(*$
<p>This function configures a generic <a target="_blank" href="#iol_slave">iol_slave</a> as a <strong>Sick WTB2SC - 2P3244</strong>. It allow to connect the object to the device-specific
parameters structure variable <a target="_blank" href="#iol_slave_wtb2sc_data">iol_slave_wtb2sc_data</a>.</p>
<p>This function should be called at startup only.</p>
$*)

FUNCTION iol_slave_mlg2prime_configure : VOID
VAR_IN_OUT
	data:						iol_slave_mlg2prime_data;			(*$	Parameters struct variable$*)
	CONVERSION_this:						iol_slave;						(*$ Instance to which the method applies $*)
END_VAR

VAR CONSTANT
	NULL:                                   			XWORD := 0;
END_VAR

//IF iol_slave_is_not_initialized(CONVERSION_this := CONVERSION_this)
//	OR
IF	iol_slave_is_configured(CONVERSION_this := CONVERSION_this)
THEN
	RETURN;
END_IF

(*** Start parameter configuration ***)

(* STANDARD PARAMETERS CONFIGURATION *)

iol_slave_configure_parameter(
	current_value_address := ADR(CONVERSION_this.vendor_name),
	configured_value_address := NULL,
	length := SIZEOF(CONVERSION_this.vendor_name),
	_type := ADST_STRING,
	coe_index := 16#0010,
	coe_sub_index := 16#00,
	readable := TRUE,
	writeable := FALSE,
	to_check := FALSE,
	CONVERSION_this := CONVERSION_this);

iol_slave_configure_parameter(
	current_value_address := ADR(CONVERSION_this.product_name),
	configured_value_address := NULL,
	length := SIZEOF(CONVERSION_this.product_name),
	_type := ADST_STRING,
	coe_index := 16#0012,
	coe_sub_index := 16#00,
	readable := TRUE,
	writeable := FALSE,
	to_check := FALSE,
	CONVERSION_this := CONVERSION_this);

iol_slave_configure_parameter(
	current_value_address := ADR(CONVERSION_this.product_id),
	configured_value_address := NULL,
	length := SIZEOF(CONVERSION_this.product_id),
	_type := ADST_STRING,
	coe_index := 16#0013,
	coe_sub_index := 16#00,
	readable := TRUE,
	writeable := FALSE,
	to_check := FALSE,
	CONVERSION_this := CONVERSION_this);


iol_slave_configure_parameter(
	current_value_address := ADR(CONVERSION_this.hardware_revision),
	configured_value_address := NULL,
	length := SIZEOF(CONVERSION_this.hardware_revision),
	_type := ADST_STRING,
	coe_index := 16#0016,
	coe_sub_index := 16#00,
	readable := TRUE,
	writeable := FALSE,
	to_check := FALSE,
	CONVERSION_this := CONVERSION_this);

iol_slave_configure_parameter(
	current_value_address := ADR(CONVERSION_this.firmware_revision),
	configured_value_address := NULL,
	length := SIZEOF(CONVERSION_this.firmware_revision),
	_type := ADST_STRING,
	coe_index := 16#0017,
	coe_sub_index := 16#00,
	readable := TRUE,
	writeable := FALSE,
	to_check := FALSE,
	CONVERSION_this := CONVERSION_this);


(* CUSTOM PARAMETERS CONFIGURATION *)


iol_slave_configure_parameter(
	current_value_address := ADR(data.CrossBeamEnable),
	configured_value_address := ADR(data.CrossBeamEnable),
	length := SIZEOF(data.CrossBeamEnable),
	_type := ADST_UINT8,
	coe_index := 16#0052,
	coe_sub_index :=16#0000,
	readable := TRUE,
	writeable := TRUE,
	to_check := TRUE, (* to be evaluated *)
	CONVERSION_this := CONVERSION_this);

iol_slave_configure_parameter(
	current_value_address := ADR(data.quality_of_teach),
	configured_value_address := NULL,
	length := SIZEOF(data.quality_of_teach),
	_type := ADST_UINT8,
	coe_index := 16#00E0,
	coe_sub_index :=16#00,
	readable := TRUE,
	writeable := FALSE,
	to_check := FALSE,
	CONVERSION_this := CONVERSION_this);
	
iol_slave_configure_parameter(
	current_value_address := ADR(data.teach_result),
	configured_value_address := NULL,
	length := SIZEOF(data.teach_result),
	_type := ADST_UINT8,
	coe_index := 16#0062,
	coe_sub_index :=16#00,
	readable := TRUE,
	writeable := FALSE,
	to_check := FALSE,
	CONVERSION_this := CONVERSION_this);

iol_slave_configure_parameter(
	current_value_address := ADR(data.temperature),
	configured_value_address := NULL,
	length := SIZEOF(data.temperature),
	_type := ADST_INT8,
	coe_index := 16#0099,
	coe_sub_index :=16#00,
	readable := TRUE,
	writeable := FALSE,
	to_check := FALSE,
	CONVERSION_this := CONVERSION_this);
	
iol_slave_configure_parameter(
	current_value_address := ADR(data.quality_of_run),
	configured_value_address := NULL,
	length := SIZEOF(data.quality_of_run),
	_type := ADST_UINT8,
	coe_index := 16#00E1,
	coe_sub_index :=16#00,
	readable := TRUE,
	writeable := FALSE,
	to_check := FALSE,
	CONVERSION_this := CONVERSION_this);
	
iol_slave_configure_parameter(
	current_value_address := ADR(data.system_status),
	configured_value_address := NULL,
	length := SIZEOF(data.system_status),
	_type := ADST_UINT8,
	coe_index := 16#0064,
	coe_sub_index :=16#00,
	readable := TRUE,
	writeable := FALSE,
	to_check := FALSE,
	CONVERSION_this := CONVERSION_this);
	
iol_slave_configure_parameter(
	current_value_address := ADR(data.device_status),
	configured_value_address := NULL,
	length := SIZEOF(data.device_status),
	_type := ADST_UINT8,
	coe_index := 16#0024,
	coe_sub_index :=16#00,
	readable := TRUE,
	writeable := FALSE,
	to_check := FALSE,
	CONVERSION_this := CONVERSION_this);
	
iol_slave_configure_parameter(
	current_value_address := ADR(data.blanking_teach_enable),
	configured_value_address := ADR(data.blanking_teach_enable),
	length := SIZEOF(data.blanking_teach_enable),
	_type := ADST_UINT8,
	coe_index := 16#0046,
	coe_sub_index :=16#00,
	readable := TRUE,
	writeable := TRUE,
	to_check := TRUE,
	CONVERSION_this := CONVERSION_this);


CONVERSION_this.CONVERSION_private.last_info_data_index := 5;

(*** End parameter configuration ***)

iol_slave_configuration_completed(
	parameters_ptr := ADR(data),
	parameters_struct_size := SIZEOF(data),
	CONVERSION_this := CONVERSION_this);

END_FUNCTION

(* stored: Version 1.1.0.1, ProductVersion 3.1.4024.3
   POU iol_slave_mlg2prime_configure: Id {b17c9068-a08e-0f8d-04c8-6e835525ece6}, SpecialFunc None *)
